// TIA Portal V20 export
DATA_BLOCK "HmiInterface"   // DB206
// stored: Access Published, MemoryReserve 100, Namespace Unit1
   VAR
      AutoStartEnable : Bool;
      InitializeEnable : Bool;
      cmFFU_LIU117 : "LER_typeLIU117Interface";
   END_VAR
   VAR RETAIN
      FFU_SleepModeRunPct : Real;
   END_VAR
   VAR
      allBrakeTest : "LER_typeBrakeTestUnitInterface";
   END_VAR
   VAR RETAIN
      BA030 : "LER_typeCommunicationInterface";
      BA040 : "LER_typeCommunicationInterface";
   END_VAR
   VAR
      BA100 { S7_SetPoint := 'True'} : "LER_typeCommunicationInterface";
   END_VAR
   VAR RETAIN
      CoveyorA : "LER_typeCommunicationInterface";
   END_VAR
BEGIN
END_DATA_BLOCK
